% RSLogix 500 project PROJECT2.RSS, saved by version 8.30.00.16 %
PROJECT "PROJECT1"    % processor: Bul.1763 MicroLogix 1100 Series B %

PROGRAM FILES
  LAD 2   3 rungs

DATA FILES
  O0 OUTPUT  4 elements
  I1 INPUT  6 elements
  S2 STATUS  66 elements
  B3 BINARY  1 elements
  T4 TIMER  1 elements
  C5 COUNTER  1 elements
  R6 CONTROL  1 elements
  N7 INTEGER  1 elements
  F8 FLOAT  1 elements

LADDER 2
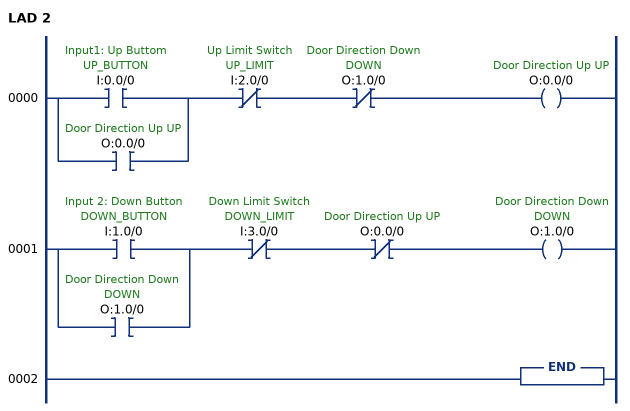
% Rung: 0 %  % edit flag set %
SOR BST XIC I:0.0/0 NXB XIC O:0.0/0 BND XIO I:2.0/0 XIO O:1.0/0 OTE O:0.0/0 EOR
%   I:0.0/0  UP_BUTTON  "Input1: Up Buttom" %
%   O:0.0/0  UP  "Door Direction Up" %
%   I:2.0/0  UP_LIMIT  "Up Limit Switch" %
%   O:1.0/0  DOWN  "Door Direction Down" %
% Rung: 1 %  % edit flag set %
SOR BST XIC I:1.0/0 NXB XIC O:1.0/0 BND XIO I:3.0/0 XIO O:0.0/0 OTE O:1.0/0 EOR
%   I:1.0/0  DOWN_BUTTON  "Input 2: Down Button" %
%   O:1.0/0  DOWN  "Door Direction Down" %
%   I:3.0/0  DOWN_LIMIT  "Down Limit Switch" %
%   O:0.0/0  UP  "Door Direction Up" %
% Rung: 2 %
SOR END EOR

OTHER DOCUMENTED ADDRESSES
  I:4.0/0  STOP  "Stop Button"
